INTERFACE I_WashStrategy

METHOD GetDuration : TIME
END_METHOD

METHOD GetRinseCount : INT
VAR_INPUT
END_VAR
END_METHOD

METHOD StartSpin : BOOL
VAR_INPUT
END_VAR
END_METHOD

METHOD StartWash : BOOL
VAR_INPUT
	iMotor : I_Motor;
END_VAR
END_METHOD

METHOD Stop
VAR_INPUT
END_VAR
END_METHOD

END_INTERFACE

(* stored: Version 1.1.0.1, ProductVersion 3.1.4024.16
   Itf I_WashStrategy: Id {6c2c2703-ab12-4238-99e3-cc10feaf744e}
   Method GetDuration: Id {4f214b80-74b8-4b0b-a1e0-7484f2ccb3ff}
   Method GetRinseCount: Id {d1479411-9084-463d-9218-d4168bf7208e}
   Method StartSpin: Id {fbca942d-b036-4ba4-a09d-4d9eaf80a064}
   Method StartWash: Id {8dab1351-8746-429b-81bf-0dda65a2482f}
   Method Stop: Id {08bd247e-b3d3-42fe-b628-1d39af0f0cac} *)
